{attribute addProperty BoxType "KL2904"}
{attribute addProperty Id "Channel_1Channel_D8611DE600"}
{attribute addProperty CRC "1578653816"}
{attribute addProperty SizeInBites "0"}
{attribute addProperty SizeInBytes "0"}
TYPE KL2904_5E185878 :
STRUCT
	{attribute addProperty Name "Channel_1"}
	Channel_1 : Channel_D8611DE6;
END_STRUCT
END_TYPE

(* stored: Version 1.2.0.0, ProductVersion 3.1.4024.9
   DUT KL2904_5E185878: Id {233b19a0-476a-4606-b9de-f6df0e580a86} *)
